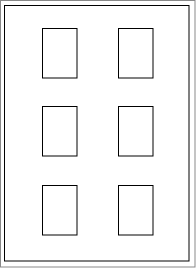
VISUALIZATION Carrinho_2  // 196x268
    RoundedRectangle (4,5 185x256)
    RoundedRectangle (35,36 50x35), angle 90, colour variable: GVL_P.corPosReator2[4].color
        OnMouseUp: execute { gvl.actReat:= 4; posCarrinho2(); }
        OnMouseUp: OpenDialog Dialog=ConfigPosicao_Reator_2, Parameters={bReator: , iOFnumber: , iSrlNumber: }, OpenModal=True, OpenCentered=True
    RoundedRectangle (111,36 50x35), angle 90, colour variable: GVL_P.corPosReator2[1].color
        OnMouseUp: OpenDialog Dialog=ConfigPosicao_Reator_2, Parameters={bReator: , iOFnumber: , iSrlNumber: }, OpenModal=True, OpenCentered=True
        OnMouseUp: execute { gvl.actReat:= 1; posCarrinho2(); }
    RoundedRectangle (111,114 50x35), angle 90, colour variable: GVL_P.corPosReator2[2].color
        OnMouseUp: execute { gvl.actReat:= 2; posCarrinho2(); }
        OnMouseUp: OpenDialog Dialog=ConfigPosicao_Reator_2, Parameters={bReator: , iOFnumber: , iSrlNumber: }, OpenModal=True, OpenCentered=True
    RoundedRectangle (35,114 50x35), angle 90, colour variable: GVL_P.corPosReator2[5].color
        OnMouseUp: execute { gvl.actReat:= 5; posCarrinho2(); }
        OnMouseUp: OpenDialog Dialog=ConfigPosicao_Reator_2, Parameters={bReator: , iOFnumber: , iSrlNumber: }, OpenModal=True, OpenCentered=True
    RoundedRectangle (111,193 50x35), angle 90, colour variable: GVL_P.corPosReator2[3].color
        OnMouseUp: execute { gvl.actReat:= 3; posCarrinho2(); }
        OnMouseUp: OpenDialog Dialog=ConfigPosicao_Reator_2, Parameters={bReator: , iOFnumber: , iSrlNumber: }, OpenModal=True, OpenCentered=True
    RoundedRectangle (35,193 50x35), angle 90, colour variable: GVL_P.corPosReator2[6].color
        OnMouseUp: execute { gvl.actReat:= 6; posCarrinho2(); }
        OnMouseUp: OpenDialog Dialog=ConfigPosicao_Reator_2, Parameters={bReator: , iOFnumber: , iSrlNumber: }, OpenModal=True, OpenCentered=True
END_VISUALIZATION

(* stored: Version 1.1.0.1, ProductVersion 3.1.4024.12
   Visu Carrinho_2: Id {773dff0d-0525-4996-81cd-7ddba10fb3ed} *)
